FUNCTION_BLOCK FB_StateMachine EXTENDS FB_DeviceBase
VAR_INPUT
    cfgAutoRun : BOOL;
    inpShutdownConfirmed : BOOL; // Application confirmation required to reset a failed Abort.
    cfgHome : ST_Permissive_Config;
    cfgStart : ST_Permissive_Config;
    cfgProceed : ST_Permissive_Config;
    cfgAuto : ST_Permissive_Config;
    cfgRunning : ST_Interlock_Config;
    inpSubmoduleFaulted : BOOL;
END_VAR

VAR_OUTPUT
    Status : ST_SM_Status;
END_VAR

VAR CONSTANT
    HOMING_MIN   : DINT := 1000; HOMING_MAX   : DINT := 1999;
    RUNNING_MIN  : DINT := 3000; RUNNING_MAX  : DINT := 3999;
    STOPPING_MIN : DINT := 2000; STOPPING_MAX : DINT := 2999;
    ABORTING_MIN : DINT := 5000; ABORTING_MAX : DINT := 5999;
    PAUSING_MIN  : DINT := 4000; PAUSING_MAX  : DINT := 4999;
    PROCEEDING_MIN : DINT := 6000; PROCEEDING_MAX : DINT := 6999;
END_VAR

VAR
    // Internal command request flags (set by methods, consumed by body)
    _abortRequested : BOOL;
    _completeStateRequested : BOOL;
    _homeRequested : BOOL;
    _pauseRequested : BOOL;
    _proceedRequested : BOOL;
    _startRequested : BOOL;
    _stopRequested : BOOL;
    _retryActive : BOOL;
    RetryComplete : BOOL;

    // OEE condition latches. Updated by ReportBlocked / ReportStarved, consumed
    // and cleared by the body each cycle. Kept internal so the FB contract
    // never mutates external inputs.
    _blockedCode : DINT;
    _starvedCode : DINT;

    // Timer
    StepTimer : TON;

    // Edge detection
    R_TRIG_1 : R_TRIG;

    // Internal state tracking
    _previousState : E_SM_State;
    PreviousStep : DINT;
    TimerReset : BOOL;
    LsOdd : DINT;
    _returnState : E_SM_State;
    ReturnNextStep : DINT;

    // Permission handlers
    permAuto : FB_Permissives;
    permHome : FB_Permissives;
    permProceed : FB_Permissives;
    permStart : FB_Permissives;

    // Running interlock (latching - auto-aborts from any active state)
    intlkRunning : FB_Interlock;

    // Step ownership (internal)
    _nextStep : DINT;
    _coverageStep : DINT := -1;
    _activeStepCalls : UINT;
    _stepFailurePending : BOOL;
    _stepRecoveryPending : BOOL;
END_VAR

_ProcessOperatorCommands();

//-----------------------------------------------------------------------------
// Main Implementation
//-----------------------------------------------------------------------------
//-------------------------------------------------------------------------
// Process permissions for different states
//-------------------------------------------------------------------------
permHome(cfg := cfgHome);
permStart(cfg := cfgStart);
permProceed(cfg := cfgProceed);
permAuto(cfg := cfgAuto);

intlkRunning(cfg := cfgRunning);
    IF inpSubmoduleFaulted THEN
        _Raise(
            code   := E_SM_Fault.SubmoduleFaulted,
            source := 'SUBMODULE',
            reason := 'Submodule reported fault via inpSubmoduleFaulted'
        );
    END_IF;
IF inpSubmoduleFaulted AND Status.State <> E_SM_State.STOPPED AND Status.State <> E_SM_State.ABORTING THEN _abortRequested := TRUE; END_IF;


    // Auto-abort if any running interlock trips (e-stop, safety gate, etc.)
    IF NOT intlkRunning.sts.bOK AND
       NOT (Status.State = E_SM_State.STOPPED OR Status.State = E_SM_State.ABORTING) THEN
        _abortRequested := TRUE;
        _Raise(
            code   := E_SM_Fault.RunningInterlockTripped,
            source := 'INTLK_RUNNING',
            reason := 'Running interlock tripped, auto-aborting'
        );
    END_IF;

    // Observe the completed application scan before consuming another transition.
    IF _coverageStep = Status.Step.Current AND Status.ActiveState AND
       Status.Step.Current MOD 2 = 0 AND NOT _stepFailurePending AND
       (NOT IsFaulted() OR Status.State = E_SM_State.STOPPING OR Status.State = E_SM_State.ABORTING) THEN
        IF _activeStepCalls = 0 THEN
            _RaiseStepFault(stepNum := Status.Step.Current, stepName := Status.Step.Name,
                code := E_SM_Fault.MissingStepImplementation, reason := 'Active FB_Step was not called in the application scan');
        ELSIF _activeStepCalls > 1 THEN
            _RaiseStepFault(stepNum := Status.Step.Current, stepName := Status.Step.Name,
                code := E_SM_Fault.DuplicateStepImplementation, reason := 'Active step was executed more than once in the application scan');
        END_IF;
    END_IF;
    _activeStepCalls := 0;

    _previousState := Status.State;
    // Sequence completion is a zero next-step requested from a valid active step.
    _completeStateRequested := _IsStepInStateRange(state := Status.State, nStep := Status.Step.Current) AND _nextStep = 0;
    Status.AutoCycleRequest := cfgAutoRun AND Status.State = E_SM_State.READY AND Status.LastState = E_SM_State.RUNNING AND NOT permStart.sts.bOK;

    // One transition per scan. Abort > Stop > fault recovery > normal transition.
    IF _stepFailurePending AND Status.State = E_SM_State.ABORTING THEN
        Status.State := E_SM_State.STOPPED;
        Status.ShutdownFailed := TRUE;
        _Raise(code := E_SM_Fault.ShutdownFailed, source := 'ABORT', reason := 'Abort sequence failed; physical shutdown confirmation required');
    ELSIF _abortRequested OR (_stepFailurePending AND Status.State = E_SM_State.STOPPING) THEN
        IF Status.State <> E_SM_State.STOPPED AND Status.State <> E_SM_State.ABORTING THEN
            Status.State := E_SM_State.ABORTING;
        END_IF;
    ELSIF _stopRequested THEN
        IF Status.State = E_SM_State.READY THEN
            Status.State := E_SM_State.STOPPED;
        ELSIF Status.State <> E_SM_State.STOPPED AND Status.State <> E_SM_State.ABORTING THEN
            Status.State := E_SM_State.STOPPING;
        END_IF;
    ELSE
        CASE Status.State OF
            E_SM_State.STOPPED:
                IF _homeRequested AND NOT IsFaulted() AND permHome.sts.bOK AND permAuto.sts.bOK AND intlkRunning.sts.bOK THEN
                    Status.State := E_SM_State.HOMING;
                END_IF;
            E_SM_State.READY:
                IF (_startRequested OR (cfgAutoRun AND Status.LastState = E_SM_State.RUNNING)) AND NOT IsFaulted() AND permStart.sts.bOK AND permAuto.sts.bOK AND intlkRunning.sts.bOK THEN
                    Status.State := E_SM_State.RUNNING;
                END_IF;
            E_SM_State.HOMING, E_SM_State.RUNNING:
                IF NOT IsFaulted() THEN
                    IF _pauseRequested AND Status.State = E_SM_State.RUNNING THEN
                        _returnState := Status.State;
                        ReturnNextStep := Status.Step.Current;
                        Status.State := E_SM_State.PAUSING;
                    ELSIF _completeStateRequested THEN
                        Status.State := E_SM_State.READY;
                    END_IF;
                END_IF;
            E_SM_State.PAUSING:
                IF _completeStateRequested AND NOT IsFaulted() THEN Status.State := E_SM_State.PAUSED; END_IF;
            E_SM_State.PAUSED:
                IF _proceedRequested AND NOT IsFaulted() AND permProceed.sts.bOK AND permAuto.sts.bOK AND intlkRunning.sts.bOK THEN
                    Status.State := E_SM_State.PROCEEDING;
                END_IF;
            E_SM_State.PROCEEDING:
                IF _completeStateRequested AND NOT IsFaulted() THEN Status.State := _returnState; END_IF;
            E_SM_State.STOPPING, E_SM_State.ABORTING:
                IF _completeStateRequested THEN Status.State := E_SM_State.STOPPED; END_IF;
        END_CASE;
    END_IF;
    IF Status.State <> _previousState THEN
        _stepFailurePending := FALSE;
        _stepRecoveryPending := FALSE;
        _ClearStepPermissives();
        Status.Step.Name := '';
        IF _previousState = E_SM_State.PROCEEDING AND Status.State = _returnState THEN
            _nextStep := ReturnNextStep;
        ELSE
            _nextStep := _GetFirstStepForState(state := Status.State);
        END_IF;
    END_IF;

    //-------------------------------------------------------------------------
    // Track state changes
    //-------------------------------------------------------------------------
    IF Status.State <> _previousState THEN
        Status.LastState := _previousState;
    END_IF;

    //-------------------------------------------------------------------------
    // Derived status flags
    //-------------------------------------------------------------------------
    Status.WaitingState := (Status.State = E_SM_State.STOPPED) OR (Status.State = E_SM_State.READY) OR
                           (Status.State = E_SM_State.PAUSED);
    Status.ActiveState  := (Status.State = E_SM_State.HOMING) OR (Status.State = E_SM_State.RUNNING) OR
                           (Status.State = E_SM_State.STOPPING) OR (Status.State = E_SM_State.PAUSING) OR
                           (Status.State = E_SM_State.PROCEEDING) OR (Status.State = E_SM_State.ABORTING);

    //-------------------------------------------------------------------------
    // Step and timer management
    //-------------------------------------------------------------------------

    // Reset timer and clear step name when transitioning to step 0
    R_TRIG_1(CLK := Status.Step.Current = 0);
    IF R_TRIG_1.Q THEN
        Status.Step.Name := '';
        _ClearStepPermissives();
        TimerReset := TRUE;
        StepTimer(IN := FALSE, PT := T#99H);
        Status.Step.TimerSeconds := 0.0;
    END_IF;

    // Auto-initialize first step when entering an active state
    IF Status.Step.Current = 0 AND Status.ActiveState THEN
        _nextStep := _GetFirstStepForState(state := Status.State);
    END_IF;

    // Detect step change and update
    IF Status.Step.Current <> _nextStep THEN
        PreviousStep := Status.Step.Current;
        Status.Step.Current := _nextStep;
        TimerReset := TRUE;
        StepTimer(IN := FALSE, PT := T#99H);
        Status.Step.TimerSeconds := 0.0;
    END_IF;

    Status.Step.Next := _nextStep;

    // Step timer logic
    IF NOT (Status.State = E_SM_State.PAUSED) OR ((Status.State = E_SM_State.PAUSED) AND _completeStateRequested) THEN
        IF TimerReset THEN
            StepTimer(IN := FALSE, PT := T#99H);
            Status.Step.TimerSeconds := 0.0;
            TimerReset := FALSE;
        ELSE
            StepTimer(IN := TRUE, PT := T#99H);
            Status.Step.TimerSeconds := UDINT_TO_REAL(TIME_TO_UDINT(StepTimer.ET)) / 1000.0;
        END_IF;
    ELSE
        StepTimer(IN := FALSE, PT := T#99H);
    END_IF;

    //-------------------------------------------------------------------------
    // Fault detection â€” surface through the shared fault handler so the
    // ring-buffer/history in ST_DeviceHeader_Sts stays populated.
    //
    // Ordering discipline:
    //   1. Submodule faults raise immediately with a specific code + source.
    //   2. OddStepReached is the "nothing more specific said anything" default
    //      for landing on an odd step. We only auto-raise it when no fault is
    //      currently active, so a more specific raise (StepTimeout raised by
    //      FB_Step, StepUserFault raised by step.RaiseFault, etc.) wins.
    //-------------------------------------------------------------------------
    LsOdd := Status.Step.Current MOD 2;
    Status.AtRecoveryStep := LsOdd <> 0;
    Status.SubmoduleFaulted := inpSubmoduleFaulted;



    IF Status.AtRecoveryStep AND GetFaultCode() = 0 THEN
        _RaiseStepFault(
            stepNum  := Status.Step.Current,
            stepName := Status.Step.Name,
            code     := E_SM_Fault.OddStepReached,
            reason   := ''
        );
    END_IF;

    //-------------------------------------------------------------------------
    // Retry logic
    //-------------------------------------------------------------------------
    IF RetryComplete THEN
        _retryActive := FALSE;
        RetryComplete := FALSE;
    END_IF;

    IF _retryActive THEN
        RetryComplete := TRUE;
    END_IF;

    IF _retryActive AND Status.AtRecoveryStep AND NOT _abortRequested AND NOT _stopRequested THEN
        // Roll back to previous (even, non-faulted) step to re-enter it
        IF NOT inpSubmoduleFaulted AND intlkRunning.sts.bOK THEN
            _ClearFault();
            _stepFailurePending := FALSE;
            _stepRecoveryPending := FALSE;
            _nextStep := Status.Step.Current - 1;
        END_IF;
    END_IF;

    //-------------------------------------------------------------------------
    // OEE condition codes (Blocked / Starved) â€” consume the internal latches.
    // The latches are fed externally via ReportBlocked() / ReportStarved().
    //-------------------------------------------------------------------------
    IF _blockedCode = 0 THEN
        Status.BlockedCondition := 0;
    END_IF;

    IF _blockedCode <> 0 AND
       (Status.State = E_SM_State.RUNNING OR Status.State = E_SM_State.STOPPING OR
        Status.State = E_SM_State.READY) THEN
        Status.BlockedCondition := _blockedCode;
        _blockedCode := 0;
    END_IF;

    IF _starvedCode = 0 THEN
        Status.StarvedCondition := 0;
    END_IF;

    IF _starvedCode <> 0 AND
       (Status.State = E_SM_State.RUNNING OR Status.State = E_SM_State.STOPPING OR
        Status.State = E_SM_State.READY) THEN
        Status.StarvedCondition := _starvedCode;
        _starvedCode := 0;
    END_IF;

    //-------------------------------------------------------------------------
    // Common device header (stateString, ready/Busy/Faulted/SourceLocked,
    // fault codes + strings, timestamps). Published via Status.header.
    //-------------------------------------------------------------------------
    Status.Faulted := IsFaulted();
    Status.ReadyToHome := Status.State = E_SM_State.STOPPED AND NOT IsFaulted() AND permHome.sts.bOK AND permAuto.sts.bOK AND intlkRunning.sts.bOK;
    Status.ReadyToStart := Status.State = E_SM_State.READY AND NOT IsFaulted() AND permStart.sts.bOK AND permAuto.sts.bOK AND intlkRunning.sts.bOK;
    Status.ReadyToProceed := Status.State = E_SM_State.PAUSED AND NOT IsFaulted() AND permProceed.sts.bOK AND permAuto.sts.bOK AND intlkRunning.sts.bOK;
    _coverageStep := Status.Step.Current;
    _ClearCommandFlags();
    _UpdateHeader(
        header      := Status.header,
        stateString := _StateToString(state := Status.State),
        busy     := Status.ActiveState
    );

METHOD PRIVATE _ClearStepPermissives
VAR
    i : UDINT;
END_VAR
Status.Step.PermCfg.nRequired := 0;
Status.Step.PermCfg.nBypassable := 0;
Status.Step.PermStatus.bOK := FALSE;
Status.Step.PermStatus.nPermissives := 0;
Status.Step.PermStatus.nBypassMask := 0;
Status.Step.PermStatus.nFirstFailureBitIndex := 999;

FOR i := 0 TO 63 DO
    Status.Step.PermCfg.aNames[i]                       := '';
    Status.Step.PermStatus.aFaceplates[i].name          := '';
    Status.Step.PermStatus.aFaceplates[i].ok         := FALSE;
    Status.Step.PermStatus.aFaceplates[i].mapped     := FALSE;
    Status.Step.PermStatus.aFaceplates[i].bypassed   := FALSE;
    Status.Step.PermStatus.aFaceplates[i].bypassable := FALSE;
END_FOR;
END_METHOD

METHOD PRIVATE _GetFirstStepForState : DINT
VAR_INPUT
        state : E_SM_State;
END_VAR
CASE state OF
        E_SM_State.HOMING:     _GetFirstStepForState := HOMING_MIN;
        E_SM_State.RUNNING:    _GetFirstStepForState := RUNNING_MIN;
        E_SM_State.STOPPING:   _GetFirstStepForState := STOPPING_MIN;
        E_SM_State.ABORTING:   _GetFirstStepForState := ABORTING_MIN;
        E_SM_State.PAUSING:    _GetFirstStepForState := PAUSING_MIN;
        E_SM_State.PROCEEDING: _GetFirstStepForState := PROCEEDING_MIN;
ELSE
        _GetFirstStepForState := 0;
END_CASE;
END_METHOD

METHOD PRIVATE _GetLastStepForState : DINT
VAR_INPUT
        state : E_SM_State;
END_VAR
CASE state OF
        E_SM_State.HOMING:     _GetLastStepForState := HOMING_MAX;
        E_SM_State.RUNNING:    _GetLastStepForState := RUNNING_MAX;
        E_SM_State.STOPPING:   _GetLastStepForState := STOPPING_MAX;
        E_SM_State.ABORTING:   _GetLastStepForState := ABORTING_MAX;
        E_SM_State.PAUSING:    _GetLastStepForState := PAUSING_MAX;
        E_SM_State.PROCEEDING: _GetLastStepForState := PROCEEDING_MAX;
ELSE
        _GetLastStepForState := 0;
END_CASE;
END_METHOD

METHOD PRIVATE _IsStepInStateRange : BOOL
VAR_INPUT
        state : E_SM_State;
        nStep : DINT;
END_VAR
_IsStepInStateRange := (_GetFirstStepForState(state := state) > 0) AND (nStep >= _GetFirstStepForState(state := state)) AND
                                             (nStep <= _GetLastStepForState(state := state));
END_METHOD

METHOD PRIVATE _StateToString : STRING(31)
VAR_INPUT
    state : E_SM_State;
END_VAR
CASE state OF
    E_SM_State.STOPPED:    _StateToString := 'STOPPED';
    E_SM_State.READY:      _StateToString := 'READY';
    E_SM_State.PAUSED:     _StateToString := 'PAUSED';
    E_SM_State.HOMING:     _StateToString := 'HOMING';
    E_SM_State.RUNNING:    _StateToString := 'RUNNING';
    E_SM_State.STOPPING:   _StateToString := 'STOPPING';
    E_SM_State.ABORTING:   _StateToString := 'ABORTING';
    E_SM_State.PAUSING:    _StateToString := 'PAUSING';
    E_SM_State.PROCEEDING: _StateToString := 'PROCEEDING';
ELSE
    _StateToString := 'UNKNOWN';
END_CASE;
END_METHOD

// Reset every pending command-request flag. Each public command method
// calls this first, then re-sets the single flag it actually requests, so
// the body only ever sees one active request at a time.
METHOD PRIVATE _ClearCommandFlags
_abortRequested         := FALSE;
_completeStateRequested := FALSE;
_homeRequested          := FALSE;
_pauseRequested         := FALSE;
_proceedRequested       := FALSE;
_startRequested         := FALSE;
_stopRequested          := FALSE;
END_METHOD

METHOD PROTECTED ResolveFaultString : STRING(79)
VAR_INPUT
    code : DINT;
END_VAR
CASE code OF
    E_SM_Fault.InvalidStepConfiguration: ResolveFaultString := 'Invalid Step Configuration';
    E_SM_Fault.MissingStepImplementation: ResolveFaultString := 'Missing Step Implementation';
    E_SM_Fault.DuplicateStepImplementation: ResolveFaultString := 'Duplicate Step Implementation';
    E_SM_Fault.ShutdownFailed: ResolveFaultString := 'Shutdown Failed';
    E_SM_Fault.None:                    ResolveFaultString := 'No Fault';
    E_SM_Fault.StepTimeout:             ResolveFaultString := 'Step Timeout';
    E_SM_Fault.OddStepReached:          ResolveFaultString := 'Step Faulted';
    E_SM_Fault.StepUserFault:           ResolveFaultString := 'Step User Fault';
    E_SM_Fault.RunningInterlockTripped: ResolveFaultString := 'Running Interlock Tripped';
    E_SM_Fault.SubmoduleFaulted:        ResolveFaultString := 'Submodule Faulted';
ELSE
    ResolveFaultString := 'Unknown Fault';
END_CASE;
END_METHOD

// Safety command â€” always accepted (bypasses source lock and fault check).
// Rejected only when the machine is already terminally stopped or already
// running the Abort sequence.
METHOD Abort : E_RpcMethodResponse
VAR_INPUT
    eRequester : E_Requester := E_Requester.PROG;
END_VAR
// Reject invalid identity before any command-specific mutation.
Abort := F_ValidateRequester(eRequester := eRequester, bSourceLocked := FALSE, bFaulted := FALSE);
IF Abort <> E_RpcMethodResponse.ACCEPTED THEN RETURN; END_IF;
IF (Status.State = E_SM_State.STOPPED AND NOT _homeRequested) OR Status.State = E_SM_State.ABORTING THEN
    Abort := E_RpcMethodResponse.REJECTED_WRONG_STATE;
    RETURN;
END_IF;

_operatorMailbox.CancelNormal();
_ClearCommandFlags();
_abortRequested := TRUE;
_retryActive := FALSE;
_AcceptCommand(eRequester := eRequester);
Abort := E_RpcMethodResponse.ACCEPTED;
END_METHOD

METHOD Home : E_RpcMethodResponse
VAR_INPUT
    eRequester : E_Requester := E_Requester.PROG;
END_VAR
// Reject invalid identity before any command-specific mutation.
Home := F_ValidateRequester(eRequester := eRequester, bSourceLocked := FALSE, bFaulted := FALSE);
IF Home <> E_RpcMethodResponse.ACCEPTED THEN RETURN; END_IF;
IF _abortRequested OR _stopRequested OR _homeRequested OR _startRequested OR _pauseRequested OR _proceedRequested THEN
    Home := E_RpcMethodResponse.REJECTED_WRONG_STATE;
    RETURN;
END_IF;
Home := F_ValidateRequester(eRequester, bSourceLockedToProg, IsFaulted());
IF Home <> E_RpcMethodResponse.ACCEPTED THEN RETURN; END_IF;

IF NOT (Status.State = E_SM_State.STOPPED) THEN
    Home := E_RpcMethodResponse.REJECTED_WRONG_STATE;
    RETURN;
END_IF;

IF NOT permHome.sts.bOK THEN
    Home := E_RpcMethodResponse.REJECTED_PERMISSIVE_NOT_MET;
    RETURN;
END_IF;

IF NOT permAuto.sts.bOK THEN
    Home := E_RpcMethodResponse.REJECTED_PERMISSIVE_NOT_MET;
    RETURN;
END_IF;

_ClearCommandFlags();
_homeRequested := TRUE;
_AcceptCommand(eRequester := eRequester);
Home := E_RpcMethodResponse.ACCEPTED;
END_METHOD

METHOD Pause : E_RpcMethodResponse
VAR_INPUT
    eRequester : E_Requester := E_Requester.PROG;
END_VAR
// Reject invalid identity before any command-specific mutation.
Pause := F_ValidateRequester(eRequester := eRequester, bSourceLocked := FALSE, bFaulted := FALSE);
IF Pause <> E_RpcMethodResponse.ACCEPTED THEN RETURN; END_IF;
IF _abortRequested OR _stopRequested OR _homeRequested OR _startRequested OR _pauseRequested OR _proceedRequested THEN
    Pause := E_RpcMethodResponse.REJECTED_WRONG_STATE;
    RETURN;
END_IF;
Pause := F_ValidateRequester(eRequester, bSourceLockedToProg, IsFaulted());
IF Pause <> E_RpcMethodResponse.ACCEPTED THEN RETURN; END_IF;

IF NOT (Status.State = E_SM_State.RUNNING) THEN
    Pause := E_RpcMethodResponse.REJECTED_WRONG_STATE;
    RETURN;
END_IF;

_ClearCommandFlags();
_pauseRequested := TRUE;
_AcceptCommand(eRequester := eRequester);
Pause := E_RpcMethodResponse.ACCEPTED;
END_METHOD

METHOD Proceed : E_RpcMethodResponse
VAR_INPUT
    eRequester : E_Requester := E_Requester.PROG;
END_VAR
// Reject invalid identity before any command-specific mutation.
Proceed := F_ValidateRequester(eRequester := eRequester, bSourceLocked := FALSE, bFaulted := FALSE);
IF Proceed <> E_RpcMethodResponse.ACCEPTED THEN RETURN; END_IF;
IF _abortRequested OR _stopRequested OR _homeRequested OR _startRequested OR _pauseRequested OR _proceedRequested THEN
    Proceed := E_RpcMethodResponse.REJECTED_WRONG_STATE;
    RETURN;
END_IF;
Proceed := F_ValidateRequester(eRequester, bSourceLockedToProg, IsFaulted());
IF Proceed <> E_RpcMethodResponse.ACCEPTED THEN RETURN; END_IF;

IF NOT (Status.State = E_SM_State.PAUSED) THEN
    Proceed := E_RpcMethodResponse.REJECTED_WRONG_STATE;
    RETURN;
END_IF;

IF NOT permProceed.sts.bOK THEN
    Proceed := E_RpcMethodResponse.REJECTED_PERMISSIVE_NOT_MET;
    RETURN;
END_IF;

IF NOT permAuto.sts.bOK THEN
    Proceed := E_RpcMethodResponse.REJECTED_PERMISSIVE_NOT_MET;
    RETURN;
END_IF;

_ClearCommandFlags();
_proceedRequested := TRUE;
_AcceptCommand(eRequester := eRequester);
Proceed := E_RpcMethodResponse.ACCEPTED;
END_METHOD

METHOD Retry : E_RpcMethodResponse
VAR_INPUT
    eRequester : E_Requester := E_Requester.PROG;
END_VAR
// Reject invalid identity before any command-specific mutation.
Retry := F_ValidateRequester(eRequester := eRequester, bSourceLocked := FALSE, bFaulted := FALSE);
IF Retry <> E_RpcMethodResponse.ACCEPTED THEN RETURN; END_IF;
// Recovery bypasses the fault gate, but never source arbitration or active interlocks.
Retry := F_ValidateRequester(eRequester, bSourceLockedToProg, FALSE);
IF Retry <> E_RpcMethodResponse.ACCEPTED THEN RETURN; END_IF;
IF _abortRequested OR _stopRequested OR NOT Status.AtRecoveryStep OR
   NOT (_stepRecoveryPending OR GetFaultCode() = E_SM_Fault.OddStepReached OR GetFaultCode() = E_SM_Fault.StepTimeout OR GetFaultCode() = E_SM_Fault.StepUserFault) THEN
    Retry := E_RpcMethodResponse.REJECTED_WRONG_STATE;
    RETURN;
END_IF;
IF inpSubmoduleFaulted OR NOT intlkRunning.sts.bOK THEN
    Retry := E_RpcMethodResponse.REJECTED_INTERLOCKED;
    RETURN;
END_IF;
_retryActive := TRUE;
_AcceptCommand(eRequester := eRequester);
Retry := E_RpcMethodResponse.ACCEPTED;
END_METHOD

METHOD Start : E_RpcMethodResponse
VAR_INPUT
    eRequester : E_Requester := E_Requester.PROG;
END_VAR
// Reject invalid identity before any command-specific mutation.
Start := F_ValidateRequester(eRequester := eRequester, bSourceLocked := FALSE, bFaulted := FALSE);
IF Start <> E_RpcMethodResponse.ACCEPTED THEN RETURN; END_IF;
IF _abortRequested OR _stopRequested OR _homeRequested OR _startRequested OR _pauseRequested OR _proceedRequested THEN
    Start := E_RpcMethodResponse.REJECTED_WRONG_STATE;
    RETURN;
END_IF;
Start := F_ValidateRequester(eRequester, bSourceLockedToProg, IsFaulted());
IF Start <> E_RpcMethodResponse.ACCEPTED THEN RETURN; END_IF;

IF NOT (Status.State = E_SM_State.READY) THEN
    Start := E_RpcMethodResponse.REJECTED_WRONG_STATE;
    RETURN;
END_IF;

IF NOT permStart.sts.bOK THEN
    Start := E_RpcMethodResponse.REJECTED_PERMISSIVE_NOT_MET;
    RETURN;
END_IF;

IF NOT permAuto.sts.bOK THEN
    Start := E_RpcMethodResponse.REJECTED_PERMISSIVE_NOT_MET;
    RETURN;
END_IF;

_ClearCommandFlags();
_startRequested := TRUE;
_AcceptCommand(eRequester := eRequester);
Start := E_RpcMethodResponse.ACCEPTED;
END_METHOD

// Safety-adjacent command â€” skip source check and fault check. Rejected only
// when the machine is already terminally stopped or already stopping.
METHOD Stop : E_RpcMethodResponse
VAR_INPUT
    eRequester : E_Requester := E_Requester.PROG;
END_VAR
// Reject invalid identity before any command-specific mutation.
Stop := F_ValidateRequester(eRequester := eRequester, bSourceLocked := FALSE, bFaulted := FALSE);
IF Stop <> E_RpcMethodResponse.ACCEPTED THEN RETURN; END_IF;
IF _abortRequested OR Status.State = E_SM_State.ABORTING OR (Status.State = E_SM_State.STOPPED AND NOT _homeRequested) OR Status.State = E_SM_State.STOPPING THEN
    Stop := E_RpcMethodResponse.REJECTED_WRONG_STATE;
    RETURN;
END_IF;

_operatorMailbox.CancelNormal();
_ClearCommandFlags();
_stopRequested := TRUE;
_retryActive := FALSE;
_AcceptCommand(eRequester := eRequester);
Stop := E_RpcMethodResponse.ACCEPTED;
END_METHOD

// External hook for OEE condition reporting. Pass a non-zero reason code while
// the machine is blocked (e.g. downstream buffer full); pass 0 to clear. The
// body publishes the active code on Status.BlockedCondition in active states.
METHOD PUBLIC ReportBlocked
VAR_INPUT
    code : DINT;
END_VAR
_blockedCode := code;
END_METHOD

// External hook for OEE condition reporting. Pass a non-zero reason code while
// the machine is starved (e.g. upstream feeder empty); pass 0 to clear.
METHOD PUBLIC ReportStarved
VAR_INPUT
    code : DINT;
END_VAR
_starvedCode := code;
END_METHOD

// Map a running interlock bit. Call every cycle. bGood=TRUE means the condition is safe.
// If bGood goes FALSE from any non-stopped state the machine auto-aborts.
METHOD MapRunningIntlk
VAR_INPUT
    bitIndex : UDINT;
    bGood    : BOOL;
END_VAR
intlkRunning.MapInput(bitIndex := bitIndex, inputValue := bGood);
END_METHOD

// Clear latched running interlock bits after the real-world condition has recovered.
// The machine will still be in STOPPED/ABORTING â€” issue Home/Start separately.
METHOD ResetRunningIntlk
intlkRunning.Reset();
END_METHOD

// INTERNAL: used by FB_Step to advance the sequence. Not part of the user API.
METHOD INTERNAL SetNextStep
VAR_INPUT
    nStep : DINT;
END_VAR
IF NOT CanExecuteStep(nStep := Status.Step.Current) THEN RETURN; END_IF;
IF nStep <> 0 AND (NOT _IsStepInStateRange(state := Status.State, nStep := nStep) OR nStep MOD 2 <> 0 OR nStep = Status.Step.Current) THEN
    _RaiseStepFault(stepNum := Status.Step.Current, stepName := Status.Step.Name,
        code := E_SM_Fault.InvalidStepConfiguration, reason := 'Destination must be zero or a different even step in the same state');
    RETURN;
END_IF;
_nextStep := nStep;
END_METHOD

// INTERNAL: used by FB_Step to publish its name to StepInfo. Not part of the user API.
METHOD INTERNAL SetStepName
VAR_INPUT
    sName : STRING(40);
END_VAR
Status.Step.Name := sName;
END_METHOD

// INTERNAL: used by FB_Step to publish the active step permissive data for HMI / OPC.
METHOD INTERNAL SetStepPermissives
VAR_INPUT
        cfg : ST_Permissive_Config;
        sts : ST_Permissive_Status;
END_VAR
Status.Step.PermCfg := cfg;
Status.Step.PermStatus := sts;
END_METHOD

// INTERNAL: unified step-fault entry point used by FB_Step (timeout, user
// RaiseFault) and by the SM body (OddStepReached auto-raise). Builds a
// default reason when the caller leaves it empty so the ring never stores
// blank context, then raises through the inherited fault book-keeping.
//
// Records the failure and selects recovery or shutdown escalation.
METHOD INTERNAL _RaiseStepFault
VAR_INPUT
    stepNum  : DINT;
    stepName : STRING(40);
    code     : DINT;
    reason   : STRING(79);
END_VAR
VAR
    effectiveCode : DINT;
    srcStr    : STRING(31);
    reasonStr : STRING(79);
END_VAR
effectiveCode := code;
IF effectiveCode <= 0 THEN effectiveCode := E_SM_Fault.StepUserFault; END_IF;
srcStr := CONCAT(STR1 := 'STEP_', STR2 := DINT_TO_STRING(stepNum));

IF reason <> '' THEN
    reasonStr := reason;
ELSE
    // Default: "Step 3004 [Advance cylinder]: Step Faulted"
    reasonStr := CONCAT(STR1 := 'Step ', STR2 := DINT_TO_STRING(stepNum));
    IF stepName <> '' THEN
        reasonStr := CONCAT(STR1 := reasonStr, STR2 := ' [');
        reasonStr := CONCAT(STR1 := reasonStr, STR2 := stepName);
        reasonStr := CONCAT(STR1 := reasonStr, STR2 := ']');
    END_IF;
    reasonStr := CONCAT(STR1 := reasonStr, STR2 := ': ');
    reasonStr := CONCAT(STR1 := reasonStr, STR2 := THIS^.ResolveFaultString(code := effectiveCode));
END_IF;

_Raise(
    code   := effectiveCode,
    source := srcStr,
    reason := reasonStr
);
Status.FailedStep := stepNum;
_stepFailurePending := TRUE;
_stepRecoveryPending := Status.State <> E_SM_State.STOPPING AND Status.State <> E_SM_State.ABORTING;
IF Status.State = E_SM_State.ABORTING THEN Status.ShutdownFailed := TRUE; END_IF;
IF _stepRecoveryPending THEN
    _nextStep := stepNum;
    IF stepNum MOD 2 = 0 THEN _nextStep := stepNum + 1; END_IF;
END_IF;
END_METHOD

METHOD PUBLIC Reset : E_RpcMethodResponse
VAR_INPUT
    eRequester : E_Requester := E_Requester.PROG;
END_VAR
// Validate identity before changing any sequence recovery state. Reset bypasses source locks.
Reset := F_ValidateRequester(eRequester := eRequester, bSourceLocked := FALSE, bFaulted := FALSE);
IF Reset <> E_RpcMethodResponse.ACCEPTED THEN RETURN; END_IF;
// Reset is recovery, not a motion-stop command. Abort/Stop first.
IF Status.State <> E_SM_State.STOPPED THEN
    Reset := E_RpcMethodResponse.REJECTED_WRONG_STATE;
    RETURN;
END_IF;
IF inpSubmoduleFaulted OR NOT intlkRunning.sts.bOK THEN
    Reset := E_RpcMethodResponse.REJECTED_INTERLOCKED;
    RETURN;
END_IF;
IF Status.ShutdownFailed AND NOT inpShutdownConfirmed THEN
    Reset := E_RpcMethodResponse.REJECTED_INTERLOCKED;
    RETURN;
END_IF;
_operatorMailbox.CancelNormal();
_stepFailurePending := FALSE;
_stepRecoveryPending := FALSE;
Status.ShutdownFailed := FALSE;
Status.FailedStep := 0;
_coverageStep := -1;
_activeStepCalls := 0;
_ClearCommandFlags();
_retryActive := FALSE;
RetryComplete := FALSE;
_nextStep := 0;
Status.Step.Current := 0;
Status.AtRecoveryStep := FALSE;
Status.Faulted := FALSE;
Reset := SUPER^.Reset(eRequester := eRequester);
END_METHOD

{attribute 'TcRpcEnable' := '1'}
METHOD PUBLIC OperatorAbort : E_RpcMethodResponse

VAR_INPUT requestId : ULINT; END_VAR
OperatorAbort := _operatorMailbox.Submit(requestId := requestId, command := E_OperatorCommand.Abort, value := 0.0);
END_METHOD

{attribute 'TcRpcEnable' := '1'}
METHOD PUBLIC OperatorHome : E_RpcMethodResponse

VAR_INPUT requestId : ULINT; END_VAR
OperatorHome := _operatorMailbox.Submit(requestId := requestId, command := E_OperatorCommand.Home, value := 0.0);
END_METHOD

{attribute 'TcRpcEnable' := '1'}
METHOD PUBLIC OperatorPause : E_RpcMethodResponse

VAR_INPUT requestId : ULINT; END_VAR
OperatorPause := _operatorMailbox.Submit(requestId := requestId, command := E_OperatorCommand.Pause, value := 0.0);
END_METHOD

{attribute 'TcRpcEnable' := '1'}
METHOD PUBLIC OperatorProceed : E_RpcMethodResponse

VAR_INPUT requestId : ULINT; END_VAR
OperatorProceed := _operatorMailbox.Submit(requestId := requestId, command := E_OperatorCommand.Proceed, value := 0.0);
END_METHOD

{attribute 'TcRpcEnable' := '1'}
METHOD PUBLIC OperatorRetry : E_RpcMethodResponse

VAR_INPUT requestId : ULINT; END_VAR
OperatorRetry := _operatorMailbox.Submit(requestId := requestId, command := E_OperatorCommand.Retry, value := 0.0);
END_METHOD

{attribute 'TcRpcEnable' := '1'}
METHOD PUBLIC OperatorStart : E_RpcMethodResponse

VAR_INPUT requestId : ULINT; END_VAR
OperatorStart := _operatorMailbox.Submit(requestId := requestId, command := E_OperatorCommand.Start, value := 0.0);
END_METHOD

{attribute 'TcRpcEnable' := '1'}
METHOD PUBLIC OperatorStop : E_RpcMethodResponse

VAR_INPUT requestId : ULINT; END_VAR
OperatorStop := _operatorMailbox.Submit(requestId := requestId, command := E_OperatorCommand.Stop, value := 0.0);
END_METHOD

{attribute 'TcRpcEnable' := '1'}
METHOD PUBLIC OperatorReset : E_RpcMethodResponse
VAR_INPUT requestId : ULINT; END_VAR
OperatorReset := _operatorMailbox.Submit(requestId := requestId, command := E_OperatorCommand.Reset, value := 0.0);
END_METHOD

METHOD PUBLIC MapHomeCondition
VAR_INPUT
    bitIndex : UDINT;
    bGood : BOOL;
END_VAR
permHome.MapInput(bitIndex := bitIndex, inputValue := bGood);
END_METHOD

METHOD PUBLIC MapStartCondition
VAR_INPUT
    bitIndex : UDINT;
    bGood : BOOL;
END_VAR
permStart.MapInput(bitIndex := bitIndex, inputValue := bGood);
END_METHOD

METHOD PUBLIC MapProceedCondition
VAR_INPUT
    bitIndex : UDINT;
    bGood : BOOL;
END_VAR
permProceed.MapInput(bitIndex := bitIndex, inputValue := bGood);
END_METHOD

METHOD PUBLIC MapAutoCondition
VAR_INPUT
    bitIndex : UDINT;
    bGood : BOOL;
END_VAR
permAuto.MapInput(bitIndex := bitIndex, inputValue := bGood);
END_METHOD

METHOD INTERNAL ObserveStep
VAR_INPUT nStep : DINT; END_VAR
IF nStep = Status.Step.Current AND nStep MOD 2 = 0 AND Status.ActiveState THEN
    IF _activeStepCalls < 2 THEN _activeStepCalls := _activeStepCalls + 1; END_IF;
END_IF;
END_METHOD

METHOD INTERNAL CanExecuteStep : BOOL
VAR_INPUT nStep : DINT; END_VAR
CanExecuteStep := nStep = Status.Step.Current AND nStep MOD 2 = 0 AND
    _IsStepInStateRange(state := Status.State, nStep := nStep) AND
    NOT _stepFailurePending AND NOT Status.ShutdownFailed AND
    (NOT IsFaulted() OR Status.State = E_SM_State.STOPPING OR Status.State = E_SM_State.ABORTING);
END_METHOD

METHOD INTERNAL ValidateStep : BOOL
VAR_INPUT nStep : DINT; nDestination : DINT; nTimeout : DINT; END_VAR
ValidateStep := nTimeout >= 0 AND nTimeout <= 356400 AND (nDestination = 0 OR
    (_IsStepInStateRange(state := Status.State, nStep := nDestination) AND nDestination MOD 2 = 0 AND nDestination <> nStep));
IF NOT ValidateStep THEN
    _RaiseStepFault(stepNum := nStep, stepName := Status.Step.Name,
        code := E_SM_Fault.InvalidStepConfiguration, reason := 'Invalid timeout or destination; use zero or another even step in this state');
END_IF;
END_METHOD

METHOD PROTECTED _DispatchOperatorCommand : E_RpcMethodResponse
VAR_INPUT command : E_OperatorCommand; value : REAL; END_VAR
CASE command OF
E_OperatorCommand.Home: _DispatchOperatorCommand := THIS^.Home(eRequester := E_Requester.OPERATOR);
E_OperatorCommand.Start: _DispatchOperatorCommand := THIS^.Start(eRequester := E_Requester.OPERATOR);
E_OperatorCommand.Stop: _DispatchOperatorCommand := THIS^.Stop(eRequester := E_Requester.OPERATOR);
E_OperatorCommand.Abort: _DispatchOperatorCommand := THIS^.Abort(eRequester := E_Requester.OPERATOR);
E_OperatorCommand.Pause: _DispatchOperatorCommand := THIS^.Pause(eRequester := E_Requester.OPERATOR);
E_OperatorCommand.Proceed: _DispatchOperatorCommand := THIS^.Proceed(eRequester := E_Requester.OPERATOR);
E_OperatorCommand.Retry: _DispatchOperatorCommand := THIS^.Retry(eRequester := E_Requester.OPERATOR);
ELSE _DispatchOperatorCommand := SUPER^._DispatchOperatorCommand(command := command, value := value);
END_CASE;
END_METHOD

END_FUNCTION_BLOCK

(* stored: Version 1.1.0.1, ProductVersion 3.1.4026.12
   POU FB_StateMachine: Id {7408693c-f749-4b9e-8684-bfcba9889df8}, SpecialFunc None
   Folder Public: Id {f0c10001-0001-0001-0001-000000000001}
   Folder Internal: Id {f0c10002-0001-0001-0001-000000000002}
   Folder Private: Id {f0c10003-0001-0001-0001-000000000003}
   Method _ClearStepPermissives: Id {d4e5f6a7-b8c9-0123-def0-123456789abf}
   Method _GetFirstStepForState: Id {d4e5f6a7-b8c9-0123-def0-123456789ac0}
   Method _GetLastStepForState: Id {d4e5f6a7-b8c9-0123-def0-123456789ac1}
   Method _IsStepInStateRange: Id {d4e5f6a7-b8c9-0123-def0-123456789ac2}
   Method _StateToString: Id {d4e5f6a7-b8c9-0123-def0-123456789ac3}
   Method _ClearCommandFlags: Id {d4e5f6a7-b8c9-0123-def0-123456789ac5}
   Method ResolveFaultString: Id {d4e5f6a7-b8c9-0123-def0-123456789ac4}
   Method Abort: Id {c1234567-1234-1234-1234-12345678C001}
   Method Home: Id {c1234567-1234-1234-1234-12345678C002}
   Method Pause: Id {c1234567-1234-1234-1234-12345678C003}
   Method Proceed: Id {c1234567-1234-1234-1234-12345678C004}
   Method Retry: Id {c1234567-1234-1234-1234-12345678C005}
   Method Start: Id {c1234567-1234-1234-1234-12345678C006}
   Method Stop: Id {c1234567-1234-1234-1234-12345678C007}
   Method ReportBlocked: Id {c1234567-1234-1234-1234-12345678C008}
   Method ReportStarved: Id {c1234567-1234-1234-1234-12345678C009}
   Method MapRunningIntlk: Id {f7a8b9c0-d1e2-4f30-a001-000000000001}
   Method ResetRunningIntlk: Id {f7a8b9c0-d1e2-4f30-a001-000000000002}
   Method SetNextStep: Id {d4e5f6a7-b8c9-0123-def0-123456789abc}
   Method SetStepName: Id {d4e5f6a7-b8c9-0123-def0-123456789abd}
   Method SetStepPermissives: Id {d4e5f6a7-b8c9-0123-def0-123456789abe}
   Method _RaiseStepFault: Id {e5f6a7b8-c9d0-1234-ef01-23456789abcd}
   Method Reset: Id {e3428cdf-4c30-4622-9cc9-dcfffe714237}
   Method OperatorAbort: Id {14e234d9-81ce-41d7-9d9b-4bda26b600ec}
   Method OperatorHome: Id {3d4f7940-8e4f-4367-8594-1371f0e9e8d6}
   Method OperatorPause: Id {b73416f4-e989-4fb7-94b3-5879a533c599}
   Method OperatorProceed: Id {1923ba34-7548-4297-88f1-c653106ed504}
   Method OperatorRetry: Id {5fd86f8d-e662-4b1b-a02c-7a65e78a9b2a}
   Method OperatorStart: Id {ee9918dd-7110-4a2f-a09e-ed4f5eb72a0b}
   Method OperatorStop: Id {5f34b2b6-c0be-419b-81e4-95c7c9bff0d7}
   Method OperatorReset: Id {d6bcf70b-4a1c-4172-a1d2-3b301484bf1a}
   Method MapHomeCondition: Id {52800701-ffb5-45c4-95f3-dd44f86fadd3}
   Method MapStartCondition: Id {441fed99-ca32-4472-bdc0-6d7325b9479d}
   Method MapProceedCondition: Id {0739f79f-49f5-4453-9a6e-fe3ebfdd13e6}
   Method MapAutoCondition: Id {c27b26eb-13d3-47f4-97cd-35e4c018c095}
   Method ObserveStep: Id {08387e71-9d75-4f3e-8f78-0828f599f1fe}
   Method CanExecuteStep: Id {a29ed26f-3dda-4e67-8817-db5c4f0a3b29}
   Method ValidateStep: Id {f041e985-e58b-4828-b9c7-fc929ca8b7b7}
   Method _DispatchOperatorCommand: Id {bb32157f-136c-4f9a-aea0-16e72a81cd44} *)
